// TIA Portal V17 export
// export: Created 2024-09-02T12:50:40.9753078Z, ExportSetting WithDefaults, DisplayName Totally Integrated Automation Portal, DisplayVersion V17, DisplayName TIA Portal Openness, DisplayVersion V17, DisplayName TIA Portal Version Control Interface, DisplayVersion V17, DisplayName STEP 7 Professional, DisplayVersion V17, DisplayName STEP 7 Safety, DisplayVersion V17, DisplayName WinCC Professional, DisplayVersion V17
TYPE "Aveva_Specyfication_WorkAuthorization"
// stored: IsFailsafeCompliant false
   STRUCT
      General : Int;   // Work authorization on the workstation: 0 = By-pass Workstation, 1 = Authorization to work
   END_STRUCT;
END_TYPE
